(* PLC project SafeLOGIC-1, BrAutomation SafeDESIGNER  4.4.0.0 *)
(* stored: companyURL http://www.br-automation.com, creationDateTime Thu Aug 19 09:51:01 2021 *)

PROGRAM Main

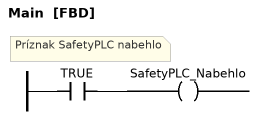
(* FBD diagram, written out as Structured Text *)
(* Príznak SafetyPLC nabehlo *)
SafetyPLC_Nabehlo := TRUE;
END_PROGRAM
